INTERFACE IService

END_INTERFACE

(* stored: Version 1.1.0.1, ProductVersion 3.1.4024.9
   Itf IService: Id {9a5b4cff-e949-4333-be56-a124fb73f4cc} *)
